(* Logix 5000 project; controller LeakTestAuto vendor 1 type 14 code 226 rev 37.11; software revision 37.01; part 15 of 15 *)
(* tags used below, declared in another part *)
   AOI_CapCylinders_Seq : AOI_Sequencer_x64;
   AOI_CapPass_Seq : AOI_Sequencer_x64;
   AOI_RobotPos : AOI_RobotPositions;
   AOI_SeqSteps : AOI_StandardSeqSteps;
   AOI_SRX100 : AOI_KeyenceBarcode;
   Barcode_ResultData : STR_Barcode;
   BarcodeBypass : BOOL;
   BarcodeInputs : udt_KeyenceScannerInputs;
   BarcodeScanner : udt_OutputStructure;
   CapCylinders_Seq : udt_SequenceStructure_X64;
   CapPass_Seq : udt_SequenceStructure_X64;
   CurrentDUTData : udt_DUTHistory[2];
   InfeedCounter : COUNTER;
   Nest1Cylinder : udt_OutputStructure;
   Nest1Ready : BOOL;
   Nest2Cylinder : udt_OutputStructure;
   Nest2Ready : BOOL;
   OP220 : udt_Mode;
   Robot : udt_OutputStructure;
   RobotGripper : udt_OutputStructure;
   RobotInputs : udt_EpsonInputs;
   TempConsumedFromPLC : BOOL;
   TON_CapCylindersDelay : TIMER;
   TON_FailChute : TIMER[10];
   I_OP220_N3_NEST1_EXTEND : ALIAS FOR Local:3:I.Pt04.Data;
   I_OP220_N3_NEST2_EXTEND : ALIAS FOR Local:3:I.Pt06.Data;
   I_OP220_N3_REJECT_BIN_OK : ALIAS FOR Local:3:I.Pt09.Data;
   I_OP220_N3_REJECT_CHUTE_PART : ALIAS FOR Local:3:I.Pt10.Data;
   OP220_EStop_OK : BOOL;
   OP220_EStopTest_DCS : DCI_STOP;
   OP220_Power : BOOL;
   PLC : AOI_PLC;
   SI_OP220_N1_CTRL_VLAVE_NC1 : ALIAS FOR Local:1:I.Pt04.Data;
   SI_OP220_N1_LASER_AREA_NC12 : ALIAS FOR Local:1:I.Pt00.Data;
   SI_OP220_N1_LASER_GUARD_NC12 : ALIAS FOR Local:1:I.Pt01.Data;
   SI_OP220_N1_SSR_12 : ALIAS FOR Local:1:I.Pt03.Data;
   SO_OP220_N2_SSR_1 : ALIAS FOR Local:2:O.Pt00.Data;
   SO_OP220_N2_SSR_2 : ALIAS FOR Local:2:O.Pt01.Data;
(* MainProgram, continued *)

ROUTINE zR60_CapCylinders   (* ladder *)
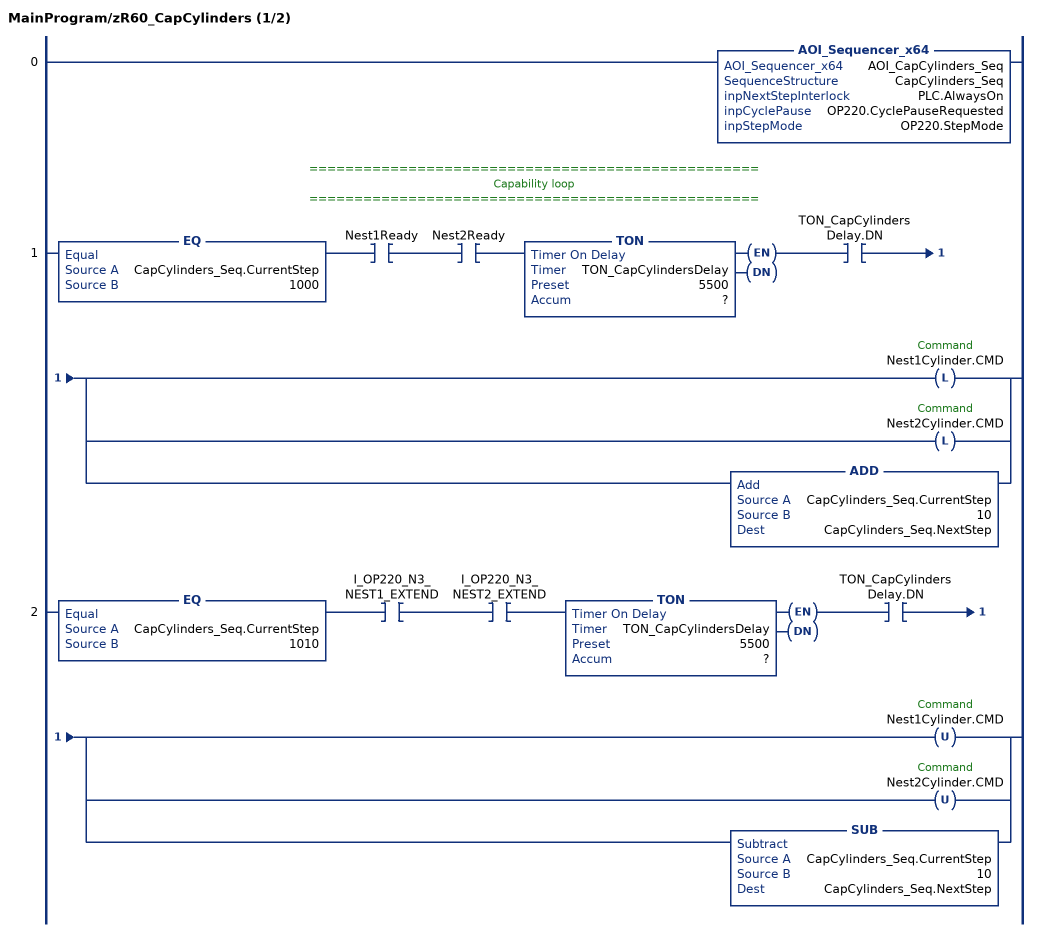
   0: AOI_Sequencer_x64(AOI_CapCylinders_Seq,CapCylinders_Seq,PLC.AlwaysOn,OP220.CyclePauseRequested,OP220.StepMode);
   // ==================================================
   // Capability loop
   // ==================================================
   1: EQ(CapCylinders_Seq.CurrentStep,1000)XIC(Nest1Ready)XIC(Nest2Ready)TON(TON_CapCylindersDelay,?,?)XIC(TON_CapCylindersDelay.DN)[OTL(Nest1Cylinder.CMD) ,OTL(Nest2Cylinder.CMD) ,ADD(CapCylinders_Seq.CurrentStep,10,CapCylinders_Seq.NextStep) ];
   2: EQ(CapCylinders_Seq.CurrentStep,1010)XIC(I_OP220_N3_NEST1_EXTEND)XIC(I_OP220_N3_NEST2_EXTEND)TON(TON_CapCylindersDelay,?,?)XIC(TON_CapCylindersDelay.DN)[OTU(Nest1Cylinder.CMD) ,OTU(Nest2Cylinder.CMD) ,SUB(CapCylinders_Seq.CurrentStep,10,CapCylinders_Seq.NextStep) ];
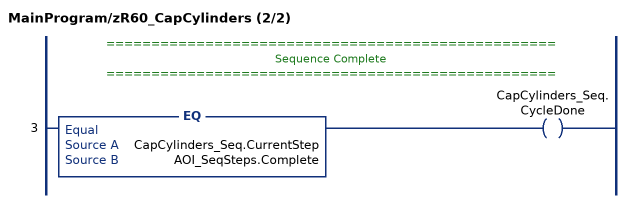
   // ==================================================
   // Sequence Complete
   // ==================================================
   3: EQ(CapCylinders_Seq.CurrentStep,AOI_SeqSteps.Complete)OTE(CapCylinders_Seq.CycleDone);
END_ROUTINE

ROUTINE zR70_CapPass   (* ladder *)
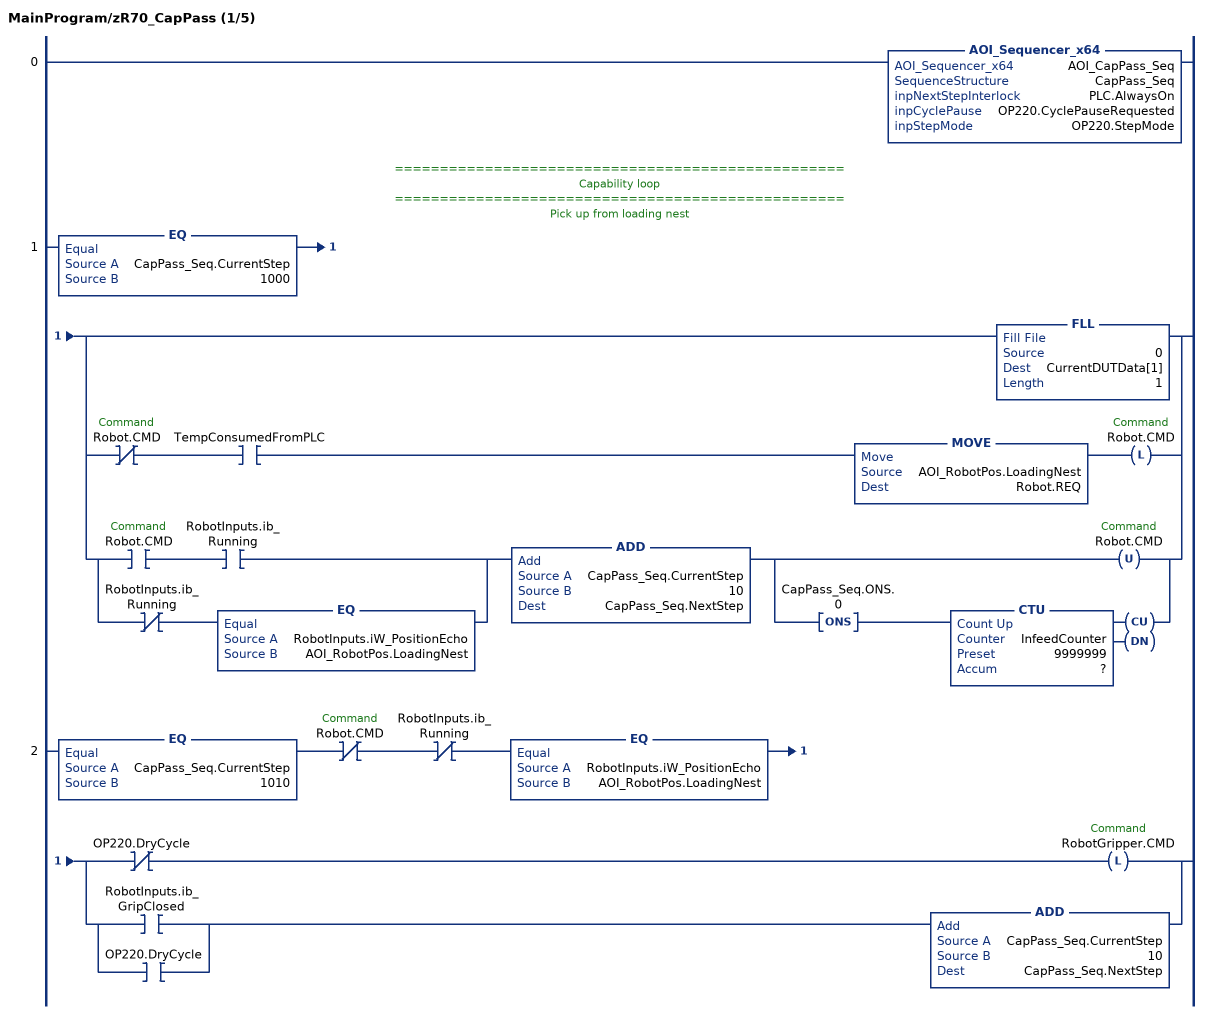
   0: AOI_Sequencer_x64(AOI_CapPass_Seq,CapPass_Seq,PLC.AlwaysOn,OP220.CyclePauseRequested,OP220.StepMode);
   // ==================================================
   // Capability loop
   // ==================================================
   // Pick up from loading nest
   1: EQ(CapPass_Seq.CurrentStep,1000)[FLL(0,CurrentDUTData[1],1) ,XIO(Robot.CMD) XIC(TempConsumedFromPLC) MOVE(AOI_RobotPos.LoadingNest,Robot.REQ) OTL(Robot.CMD) ,[XIC(Robot.CMD) XIC(RobotInputs.ib_Running) ,XIO(RobotInputs.ib_Running) EQ(RobotInputs.iW_PositionEcho,AOI_RobotPos.LoadingNest) ] ADD(CapPass_Seq.CurrentStep,10,CapPass_Seq.NextStep) [OTU(Robot.CMD) ,ONS(CapPass_Seq.ONS.0) CTU(InfeedCounter,?,?) ] ];
   2: EQ(CapPass_Seq.CurrentStep,1010)XIO(Robot.CMD)XIO(RobotInputs.ib_Running)EQ(RobotInputs.iW_PositionEcho,AOI_RobotPos.LoadingNest)[XIO(OP220.DryCycle) OTL(RobotGripper.CMD) ,[XIC(RobotInputs.ib_GripClosed) ,XIC(OP220.DryCycle) ] ADD(CapPass_Seq.CurrentStep,10,CapPass_Seq.NextStep) ];
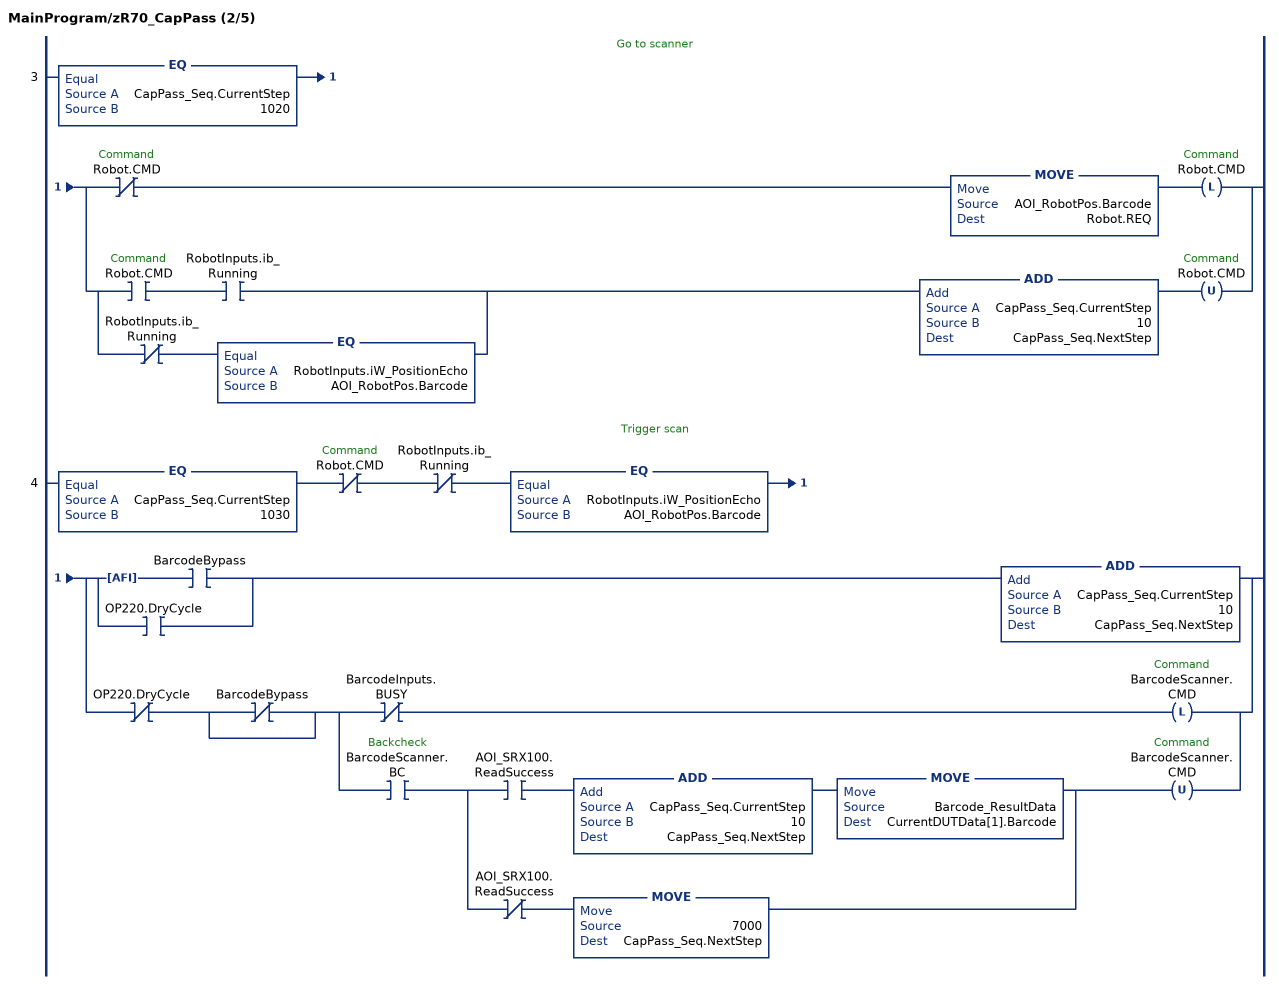
   // Go to scanner
   3: EQ(CapPass_Seq.CurrentStep,1020)[XIO(Robot.CMD) MOVE(AOI_RobotPos.Barcode,Robot.REQ) OTL(Robot.CMD) ,[XIC(Robot.CMD) XIC(RobotInputs.ib_Running) ,XIO(RobotInputs.ib_Running) EQ(RobotInputs.iW_PositionEcho,AOI_RobotPos.Barcode) ] ADD(CapPass_Seq.CurrentStep,10,CapPass_Seq.NextStep) OTU(Robot.CMD) ];
   // Trigger scan
   4: EQ(CapPass_Seq.CurrentStep,1030)XIO(Robot.CMD)XIO(RobotInputs.ib_Running)EQ(RobotInputs.iW_PositionEcho,AOI_RobotPos.Barcode)[[AFI() XIC(BarcodeBypass) ,XIC(OP220.DryCycle) ] ADD(CapPass_Seq.CurrentStep,10,CapPass_Seq.NextStep) ,XIO(OP220.DryCycle) [XIO(BarcodeBypass) ,] [XIO(BarcodeInputs.BUSY) OTL(BarcodeScanner.CMD) ,XIC(BarcodeScanner.BC) [XIC(AOI_SRX100.ReadSuccess) ADD(CapPass_Seq.CurrentStep,10,CapPass_Seq.NextStep) MOVE(Barcode_ResultData,CurrentDUTData[1].Barcode) ,XIO(AOI_SRX100.ReadSuccess) MOVE(7000,CapPass_Seq.NextStep) ] OTU(BarcodeScanner.CMD) ] ];
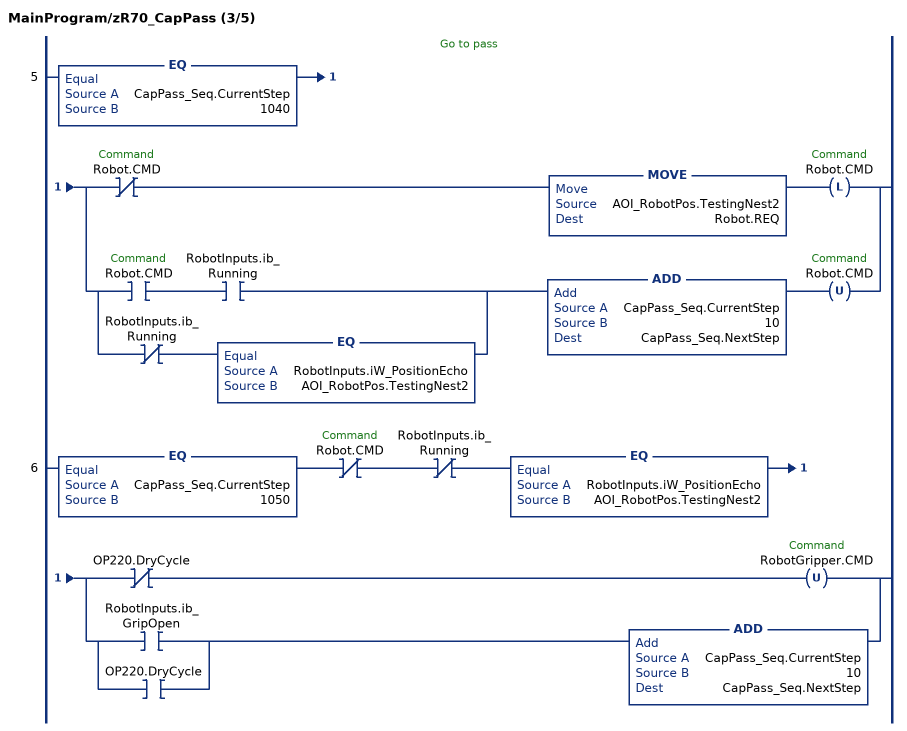
   // Go to pass
   5: EQ(CapPass_Seq.CurrentStep,1040)[XIO(Robot.CMD) MOVE(AOI_RobotPos.TestingNest2,Robot.REQ) OTL(Robot.CMD) ,[XIC(Robot.CMD) XIC(RobotInputs.ib_Running) ,XIO(RobotInputs.ib_Running) EQ(RobotInputs.iW_PositionEcho,AOI_RobotPos.TestingNest2) ] ADD(CapPass_Seq.CurrentStep,10,CapPass_Seq.NextStep) OTU(Robot.CMD) ];
   6: EQ(CapPass_Seq.CurrentStep,1050)XIO(Robot.CMD)XIO(RobotInputs.ib_Running)EQ(RobotInputs.iW_PositionEcho,AOI_RobotPos.TestingNest2)[XIO(OP220.DryCycle) OTU(RobotGripper.CMD) ,[XIC(RobotInputs.ib_GripOpen) ,XIC(OP220.DryCycle) ] ADD(CapPass_Seq.CurrentStep,10,CapPass_Seq.NextStep) ];
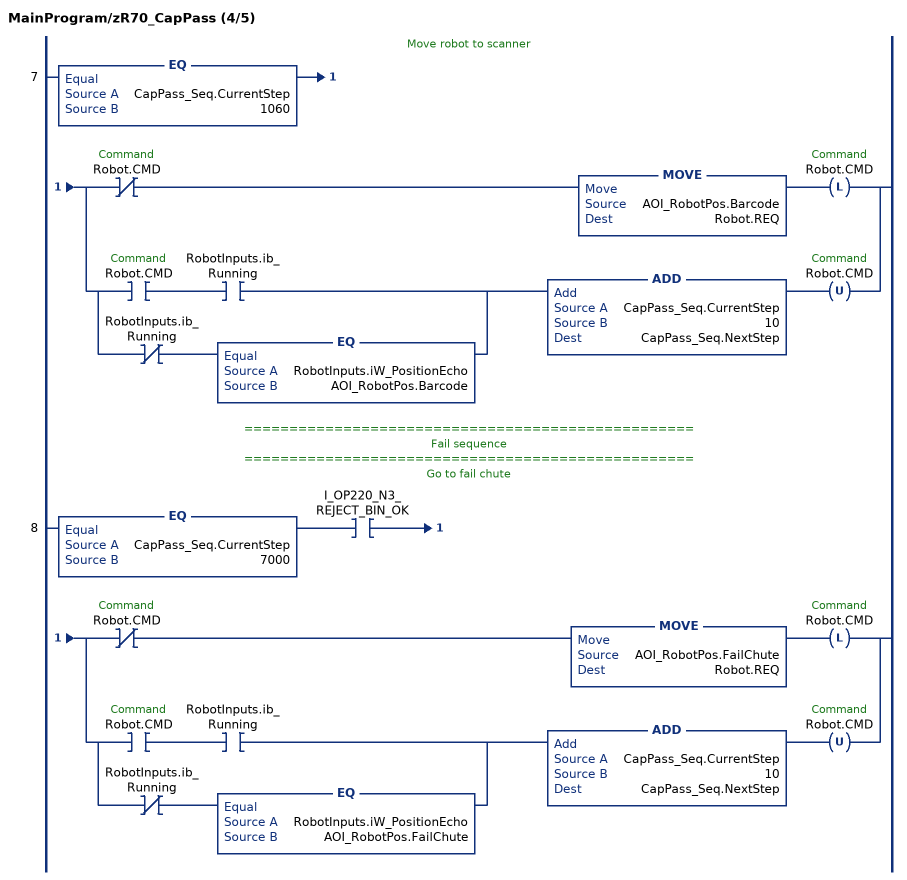
   // Move robot to scanner
   7: EQ(CapPass_Seq.CurrentStep,1060)[XIO(Robot.CMD) MOVE(AOI_RobotPos.Barcode,Robot.REQ) OTL(Robot.CMD) ,[XIC(Robot.CMD) XIC(RobotInputs.ib_Running) ,XIO(RobotInputs.ib_Running) EQ(RobotInputs.iW_PositionEcho,AOI_RobotPos.Barcode) ] ADD(CapPass_Seq.CurrentStep,10,CapPass_Seq.NextStep) OTU(Robot.CMD) ];
   // ==================================================
   // Fail sequence
   // ==================================================
   // Go to fail chute
   8: EQ(CapPass_Seq.CurrentStep,7000)XIC(I_OP220_N3_REJECT_BIN_OK)[XIO(Robot.CMD) MOVE(AOI_RobotPos.FailChute,Robot.REQ) OTL(Robot.CMD) ,[XIC(Robot.CMD) XIC(RobotInputs.ib_Running) ,XIO(RobotInputs.ib_Running) EQ(RobotInputs.iW_PositionEcho,AOI_RobotPos.FailChute) ] ADD(CapPass_Seq.CurrentStep,10,CapPass_Seq.NextStep) OTU(Robot.CMD) ];
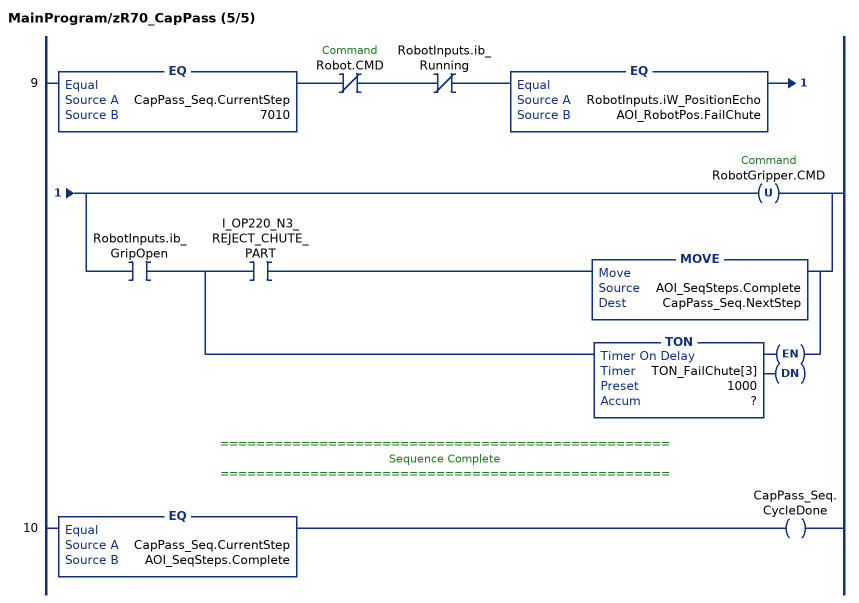
   9: EQ(CapPass_Seq.CurrentStep,7010)XIO(Robot.CMD)XIO(RobotInputs.ib_Running)EQ(RobotInputs.iW_PositionEcho,AOI_RobotPos.FailChute)[OTU(RobotGripper.CMD) ,XIC(RobotInputs.ib_GripOpen) [XIC(I_OP220_N3_REJECT_CHUTE_PART) MOVE(AOI_SeqSteps.Complete,CapPass_Seq.NextStep) ,TON(TON_FailChute[3],?,?) ] ];
   // ==================================================
   // Sequence Complete
   // ==================================================
   10: EQ(CapPass_Seq.CurrentStep,AOI_SeqSteps.Complete)OTE(CapPass_Seq.CycleDone);
END_ROUTINE

ROUTINE zzUnused   (* ladder *)
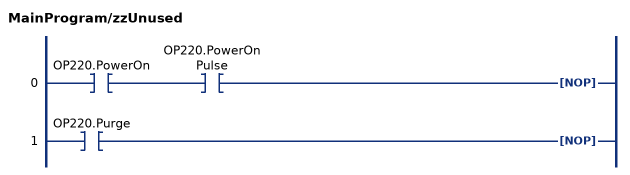
   0: XIC(OP220.PowerOn)XIC(OP220.PowerOnPulse)NOP();
   1: XIC(OP220.Purge)NOP();
END_ROUTINE
END_PROGRAM

PROGRAM SafetyProgram   (* main routine MainRoutine, safety *)
VAR
   TON_EStopFaultReset : TIMER := (PRE := 1000);
END_VAR

ROUTINE MainRoutine   (* ladder *)
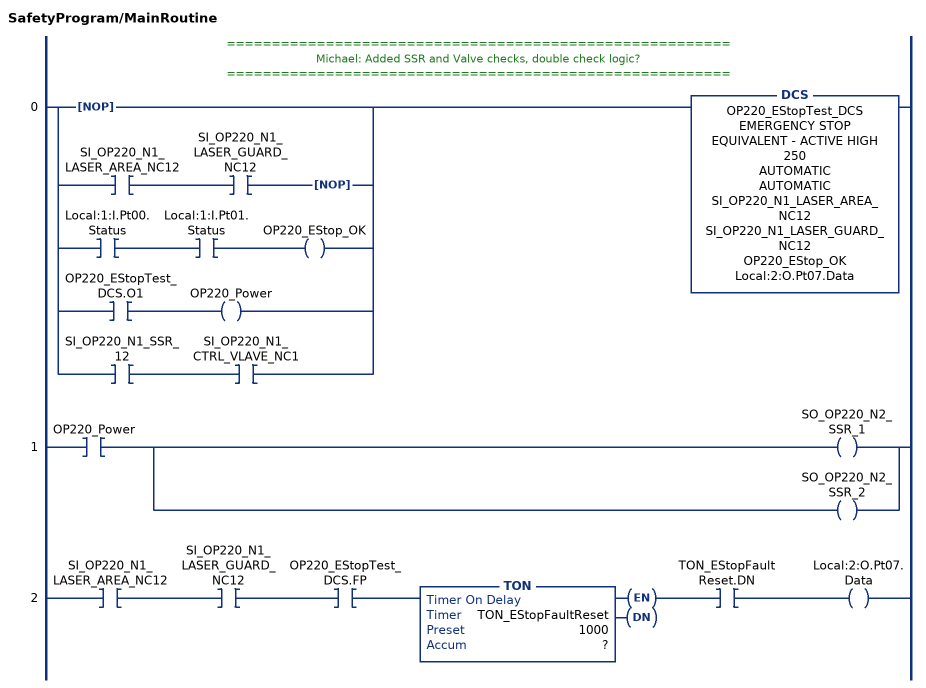
   // ========================================================
   // Michael: Added SSR and Valve checks, double check logic?
   // ========================================================
   0: [NOP() ,XIC(SI_OP220_N1_LASER_AREA_NC12) XIC(SI_OP220_N1_LASER_GUARD_NC12) NOP() ,XIC(Local:1:I.Pt00.Status) XIC(Local:1:I.Pt01.Status) OTE(OP220_EStop_OK) ,XIC(OP220_EStopTest_DCS.O1) OTE(OP220_Power) ,XIC(SI_OP220_N1_SSR_12) XIC(SI_OP220_N1_CTRL_VLAVE_NC1) ]DCS(OP220_EStopTest_DCS,EMERGENCY STOP,EQUIVALENT - ACTIVE HIGH,250,AUTOMATIC,AUTOMATIC,SI_OP220_N1_LASER_AREA_NC12,SI_OP220_N1_LASER_GUARD_NC12,OP220_EStop_OK,Local:2:O.Pt07.Data);
   1: XIC(OP220_Power)[OTE(SO_OP220_N2_SSR_1) ,OTE(SO_OP220_N2_SSR_2) ];
   2: XIC(SI_OP220_N1_LASER_AREA_NC12)XIC(SI_OP220_N1_LASER_GUARD_NC12)XIC(OP220_EStopTest_DCS.FP)TON(TON_EStopFaultReset,?,?)XIC(TON_EStopFaultReset.DN)OTE(Local:2:O.Pt07.Data);
END_ROUTINE
END_PROGRAM
